(* CODESYS project Hand_Grab_Control_blocks.export

Project tree, tasks and I/O mapping:
  Hand_Grab_Control_blocks/
    data type Gesture_Type
    data type Grab_Command
    data type Grab_State
    data type PhysicalHandType
    function block Grab_Control [ST]
    function block Grab_Demo [ST]
    function block Hand_Gesture [ST]
    function block Hand_Gesture_Demo [ST]
*)

// Hand_Grab_Control_blocks/Gesture_Type
{attribute 'qualified_only'}
{attribute 'strict'}
TYPE Gesture_Type :
(
	Gesture_Type_None			:= 0,
	Gesture_Type_Num_1		:= 1,
	Gesture_Type_Num_2		:= 2,
	Gesture_Type_Num_3		:= 3,
	Gesture_Type_Num_4		:= 4,
	Gesture_Type_Num_5		:= 5,
	Gesture_Type_Num_6		:= 6,
	Gesture_Type_Fist			:= 10,
	Gesture_Type_Palm			:= 11,
	Gesture_Type_ThumbUp		:= 12,
	Gesture_Type_NoNoNo			:= 13,
	Gesture_Type_ComeOnBaby	:= 14,
	Gesture_Type_FingerWave		:= 15,
	Gesture_Type_Wave			:= 16,
	Gesture_Type_Nya			:= 17,
	Gesture_Type_MovObj			:= 18
);
END_TYPE

// Hand_Grab_Control_blocks/Grab_Command
TYPE Grab_Command :
STRUCT
	Tip_Angle : REAL;
	Root_Angle : REAL;
	Clamp_Angle : REAL;
END_STRUCT
END_TYPE

// Hand_Grab_Control_blocks/Grab_State
TYPE Grab_State :
STRUCT
	Tip_State : BOOL;
	Root_State : BOOL;
	Clamp_Angle : REAL;
END_STRUCT
END_TYPE

// Hand_Grab_Control_blocks/PhysicalHandType
TYPE PhysicalHandType :
(
	motor18		:= 0	// total 18 motors. 4 axis for thumb, 3 axis control 2 joints, anohter one control thumb tip joint. Other fingers has 3 axis each, each axis control 1 jonit. 2 axis for each wrist joint.
	, motor17	:= 10	// total 17 motors, each axis control 1 joint.
);
END_TYPE

// Hand_Grab_Control_blocks/Grab_Control
FUNCTION_BLOCK Grab_Control
VAR_INPUT
	Enable : BOOL;
	OverFeed : INT;
	Grab : Grab_Command;
	GrabFirstAxis : BYTE;
	GrabLastAxis : BYTE;
	GrabAxisAllowToMov : ARRAY [0..2] OF BOOL;
END_VAR
VAR_OUTPUT
	Done : BOOL;
	isMoving : BOOL;
	Error : BOOL;
	Err_Message : Error_Message;
	MinClampAng : REAL;
	MaxClampAng : REAL;
	MinRootAng : REAL;
	MaxRootAng : REAL;
	MinTipAng : REAL;
	MaxTipAng : REAL;
END_VAR
VAR
	state : INT := 0;
	i : INT;
	//movment settings
	Finger_Movement: MultiAxisABSMove;
	MultiMov_for_counter : INT;
	Give_Finger_Pos_Counter : INT;
	GivHandPos : ARRAY [0..255] OF REAL;
	handVel : REAL := 402;	// 402 = 67rpm
	handAcc : REAL := 4020;
	handJerk : REAL := 40200;
	givenVel, givenAcc, givenJerk : REAL;
	ArrayTotalNum : INT;
	ArrayFirstRow : INT;
	AxisAllowToMov : ARRAY [0..255] OF BOOL;
	faxis: BYTE;	// first finge axis number
	laxis : BYTE;	// last finger axis number
	
	// grab pos
	g_grab: ARRAY [0..32] OF REAL;
	
	// max degree for every motor
	grab_angle_min : REAL := 0;
	grab_angle_max : REAL := -75; //BASE
	
	Root_min : REAL := 0;
	Root_max : REAL := -138; //TURN
	
	Tip_min : REAL := 0;
	Tip_max : REAL := -86; //ROTAR
	
	// debug
	mid_0_max: REAL;
	mid_0_min: REAL;
	
	clamp : Value_Clamp;
	_ov: REAL;
END_VAR

MinClampAng := grab_angle_min;
MaxClampAng := grab_angle_max;
MinRootAng := Root_min;
MaxRootAng := Root_max;
MinTipAng := Tip_min;
MaxTipAng := Tip_max;

IF NOT Enable AND state > 0 THEN
	state := 0;
END_IF

_ov := overfeed;
IF _ov > 100 THEN
	_ov := 100;
ELSIF _ov < 1 THEN
	_ov := 1;
END_IF

Finger_Movement(firstAuxAxisNum := faxis, LastAuxAxisNum := laxis, enable := state > 0);
CASE state OF
	-30:
		error := TRUE;
		Err_Message := error_message.Err_AuxAxis_Movement_Block_err;
	-10:
	(*
		IF ReadCurrentPos.ErrorID THEN
			
		END_IF
	*)
		error := TRUE;
		Err_Message := error_message.Err_AuxAxis_Movement_Cannot_read_virture_robot_position;
	-1:
		error := TRUE;
		// can not handle more than three axis
		
	0:
		Done := error := FALSE;
		Err_Message := error_message.Err_None;
		
		IF Enable THEN
			faxis := GrabFirstAxis;
			laxis := GrabLastAxis;
			IF (laxis - faxis) <= 2 THEN
				state := 10;
			ELSE
				state := -1;
			END_IF
		END_IF

	10:	//initialize
	
		// set position
		
		// clamp Angle
		clamp(current := Grab.Clamp_Angle, first_value := grab_angle_min, second_value := grab_angle_max, newV => g_grab[0]);
		
		// clamp Root_Angle
		clamp(current := Grab.Root_Angle, first_value := Root_min, second_value := Root_max, newV => g_grab[1]);
		
		// clamp Tip_Angle
		clamp(current := Grab.Tip_Angle, first_value := Tip_min, second_value := Tip_max, newV => g_grab[2]);
		
		
		// asign value for hand movment block
		Give_Finger_Pos_Counter := 0;
		FOR MultiMov_for_counter := faxis TO laxis DO
			AxisAllowToMov[MultiMov_for_counter] := GrabAxisAllowToMov[MultiMov_for_counter - faxis];
			GivHandPos[MultiMov_for_counter] := g_grab[Give_Finger_Pos_Counter];
			Give_Finger_Pos_Counter := Give_Finger_Pos_Counter + 1;
		END_FOR
		Finger_Movement(Execute:=FALSE);
		
		givenVel := handVel * (_ov/100.0);
		givenAcc := handAcc * (_ov/100.0);
		givenJerk := handJerk * (_ov/100.0);

		State := 20;
	20:
		Finger_Movement(execute := TRUE, Axis_Mov_Indicator := AxisAllowToMov, axis_mov_pos := GivHandPos
			, vel := givenVel, acc :=givenAcc, dec := givenAcc, jerk := givenJerk, MoveMethod := 10);
		//Finger_Movement(AxesGroup:=0, Execute:=TRUE, Position:=Pos_For_Hand_Block, Settings:=Set1, active => isMoving);
		
		IF Finger_Movement.Done THEN
			Finger_Movement(Execute:=FALSE);
			done := TRUE;
			state := 50;
		ELSIF Finger_Movement.Error THEN
			state := -30;
		END_IF
	50:
			done := TRUE;
END_CASE
// end of the program

END_FUNCTION_BLOCK

// Hand_Grab_Control_blocks/Grab_Demo
FUNCTION_BLOCK Grab_Demo
VAR_INPUT
	enable :BOOL;
	internal_hand_enable : BOOL;
	startMov :BOOL;
	ovr : INT;
	GrabFirstAxis : BYTE;
	GrabLastAxis : BYTE;
	GrabAxisAllowToMov : ARRAY [0..2] OF BOOL;
END_VAR

VAR_OUTPUT
	IsEnabled : BOOL;
	IsMoving : BOOL;
	err : BOOL;
	err_message : error_message;
END_VAR

VAR
	
	// state control
	cycleState : INT;	// state machine
	cycleCounter : INT;	// counte how many time already been done
	start_cycle : INT := -1;	// start cycle from a number
	total_cycle_time : INT := 23; //	max cycle time
	cycleTimer : ton;
	cycleDelayTime : TIME := T#0MS;	// delay time between every gesture
	
	// hand powerOn
	powerHand : BOOL;
	powerOnHand : AuxAxis_PowerOn;
	_enabled : BOOL;
	
	// gestrure mov block
	GrabMov : Grab_Control;
	GrabCmd : grab_command;
	_GrabCmdEmpt : grab_command;
END_VAR


//err
IF powerOnHand.Error OR GrabMov.Error THEN
	err := TRUE;
	IF powerOnHand.Error THEN
		err_message := powerOnHand.Err_Message;
	ELSIF GrabMov.Error THEN
		err_message := GrabMov.Err_Message;
	END_IF
ELSE
	err := FALSE;
	err_message := error_message.Err_None;
END_IF

// enable hand
IF internal_hand_enable THEN
	powerOnHand(enable := enable);
	_enabled := IsEnabled := powerOnHand.Done;
END_IF

IF _enabled AND NOT internal_hand_enable THEN
	powerOnHand(enable := internal_hand_enable);
	_enabled := IsEnabled := powerOnHand.Done;
END_IF

IF NOT enable THEN
	cycleState := 0;
	isMoving := FALSE;
	cycleTimer(in := FALSE);	// reset timer
	GrabMov(Enable := FALSE);	// reset movement block
END_IF

CASE cycleState OF
	0: 
		// if block is enabled and order to move and (manager by internal power or by external power)
		IF enable AND startMov AND (NOT internal_hand_enable OR _enabled) THEN
			GrabCmd.Root_Angle := GrabMov.minRootAng;	// all open
			GrabCmd.Tip_Angle := GrabMov.minTipAng;
			GrabCmd.Clamp_Angle := GrabMov.minClampAng;
			
			cycleCounter := start_cycle;	// set counter to start_cycle
			cycleState := 10;
		END_IF
	10:
		GrabMov(Enable := TRUE, overfeed := ovr,Grab := GrabCmd, isMoving => isMoving
				, GrabFirstAxis := GrabFirstAxis, GrabLastAxis:= GrabLastAxis, GrabAxisAllowToMov:= GrabAxisAllowToMov);
		
		IF NOT startMov THEN
			GrabMov(Enable := FALSE);
			cycleState := 0;
		END_IF
		IF GrabMov.Done THEN
			cycleTimer(in := TRUE, pt:= cycleDelayTime);	// start timer for delay
			IF cycleTimer.Q THEN	// time reach
				cycleCounter := cycleCounter + 1;	// done and self add for next gesture
				cycleTimer(in := FALSE);	// reset timer
				GrabMov(Enable := FALSE);	// reset movement block
				
				IF cycleCounter <= total_cycle_time THEN
					IF cycleCounter <= 5 THEN	// first movement, root as clamp
						IF (cycleCounter MOD 2) = 1 THEN
							GrabCmd.Root_Angle := GrabMov.minRootAng;
						ELSE
							GrabCmd.Root_Angle := GrabMov.MaxRootAng;
						END_IF
					ELSIF cycleCounter <= 11 THEN	// second movement, show tip movement
						IF (cycleCounter MOD 2) = 1 THEN
							GrabCmd.Tip_Angle := GrabMov.MinTipAng;
						ELSE
							GrabCmd.Tip_Angle := GrabMov.MaxTipAng;
						END_IF
					ELSIF cyclecounter <= 17 THEN	// second movement, tip as clamp
							GrabCmd.Root_Angle := GrabMov.MaxRootAng/2;
						IF (cycleCounter MOD 2) = 1 THEN
							GrabCmd.Tip_Angle := GrabMov.MinTipAng;
						ELSE
							GrabCmd.Tip_Angle := GrabMov.MaxTipAng;
						END_IF
					ELSIF cyclecounter <= 23 THEN	// third movement, show clamp angle
						GrabCmd.Root_Angle := GrabMov.minRootAng;
						GrabCmd.Tip_Angle := GrabMov.minTipAng;
						IF (cycleCounter MOD 2) = 1 THEN;
							GrabCmd.Clamp_Angle := GrabMov.MinClampAng;
						ELSE
							GrabCmd.Clamp_Angle := GrabMov.MaxClampAng;
						END_IF
					ELSIF cyclecounter <= 24 THEN	// fouth movement, tip as clamp in another clamp angle
					END_IF
					cycleState := 10;	// if not reach total number then go back keep do next gesture
				ELSE
					cycleState := 0;	// if reach maximum then go back beginning
				END_IF
			END_IF
		END_IF
END_CASE

END_FUNCTION_BLOCK

// Hand_Grab_Control_blocks/Hand_Gesture
FUNCTION_BLOCK Hand_Gesture
VAR_INPUT
	Enable : BOOL;
	OverFeed : INT;
	Gesture : Gesture_Type;
	HandType : PhysicalHandType;	
	HandFirstAxis : BYTE;
	HandLastAxis : BYTE;
	HandAxisAllowToMov : ARRAY [0..17] OF BOOL;
END_VAR
VAR_OUTPUT
	Done : BOOL;
	isMoving : BOOL;
	Error : BOOL;
	Err_Message : Error_Message;
END_VAR
VAR
	_enb : BOOL;
	state : INT := 0;
	i : INT;
	//movment settings
	_ov : REAL;
	FingerMovPos: ARRAY [1..32] OF REAL;
	SecFingerMovPos: ARRAY [1..32] OF REAL;
	ThdFingerMovPos: ARRAY [1..32] OF REAL;
	CycleMovTimes : INT := 1;
	CycleMovDone : BOOL;
	
	CycleFingerMovPos: ARRAY [0..20] OF ARRAY[1..32] OF REAL;	
	DelayTimer : ton;
	DelayTime : ARRAY [0..20] OF TIME;
	readyToMov : BOOL;
	G_MovObj_Muilt : INT;
	
	MultisingleMov : MultiAxisABSMove;
	MultiMov_for_counter : INT;
	Give_Finger_Pos_Counter : INT;
	GivHandPos : ARRAY [0..255] OF REAL;
	handVel : REAL := 402;	// 402 = 67rpm
	handAcc : REAL := 4020;
	handJerk : REAL := 40200;
	givenVel, givenAcc, givenJerk : REAL;
	ArrayTotalNum : INT;
	ArrayFirstRow : INT;
	ReadTorque : ARRAY [0..255] OF ArcaLibrary.MCAT_ReadAxisMeasures;
	ReadTorque_For : INT;
	HandAxisTorqueValue_Sum : ARRAY [0..255] OF REAL;
	HandAxisTorqueValue_Raw : ARRAY [0..255] OF REAL;
	HandAxisTorqueValue_Smooth: ARRAY [0..255] OF REAL;
	TorqueSmoothTime : TIME := T#2S;
	TorqueSmoothTimer : ton;
	TorqueSmoothLoopTime : BYTE;
	// gesture pos
	g_RestPos: ARRAY [1..32] OF REAL;
	g_one: ARRAY [1..32] OF REAL;
	g_two: ARRAY [1..32] OF REAL;
	g_three: ARRAY [1..32] OF REAL;
	g_four: ARRAY [1..32] OF REAL;
	g_five: ARRAY [1..32] OF REAL;
	g_six: ARRAY [1..32] OF REAL;
	g_plam: ARRAY [1..32] OF REAL;
	g_fist: ARRAY [1..32] OF REAL;
	g_thumbUp: ARRAY [1..32] OF REAL;
	
	// max degree for every motor
	wrist_0_min : REAL := 0;
	wrist_0_max : REAL := 58;
	wrist_1_min : REAL := 0;
	wrist_1_max : REAL := 58;
	
	// axis 0 to axis 2
	thumb_group_pos_0 : ARRAY[0..2] OF REAL := [000, 005, 002];		// thump relex and thump tip open
	thumb_group_pos_1 : ARRAY[0..2] OF REAL := [000, 078, 002];		// thump relex and thump tip close	// this has been used in gesture fingerwave
	thumb_group_pos_2 : ARRAY[0..2] OF REAL := [120, 005, 073];		// thumb close and thump tip open	// this has been assigned to most case when thumb need to close
	thumb_group_pos_3 : ARRAY[0..2] OF REAL := [120, 078, 073];		// thumb close and thump tip close
	thumb_3_min : REAL := 0;
	thumb_3_max : REAL := 5;
	(*
	thumb_0_min : REAL := 0;
	thumb_0_max : REAL := 120;
	thumb_1_min : REAL := 5;
	thumb_1_max : REAL := 78;
	thumb_2_min : REAL := 2;
	thumb_2_max : REAL := 73;
	*)
	
	index_0_min : REAL := 0;
	index_0_max : REAL := 20;
	index_1_min : REAL := 2;
	index_1_max : REAL := 74;
	index_2_min : REAL := 1;
	index_2_max : REAL := 87;
		
	mid_0_min : REAL := 0;
	mid_0_max : REAL := 15;
	mid_1_min : REAL := 3;
	mid_1_max : REAL := 66;
	mid_2_min : REAL := 2;
	mid_2_max : REAL := 68;
			
	ring_0_min : REAL := 0;
	ring_0_max : REAL := 10;
	ring_1_min : REAL := 2;
	ring_1_max : REAL := 53;
	ring_2_min : REAL := 2;
	ring_2_max : REAL := 68;
		
	little_0_min : REAL :=0;
	little_0_max : REAL := 20;
	little_1_min : REAL := 3;
	little_1_max : REAL := 81;
	little_2_min : REAL := 1;
	little_2_max : REAL := 78;
	
	// debug
	//temp_HandType : PhysicalHandType := motor18;
	AxisAllowToMov : ARRAY [0..255] OF BOOL;
	faxis: BYTE;	// first finge axis number
	laxis : BYTE;	// last finger axis number
END_VAR

IF NOT Enable THEN
	IF _enb THEN
		_enb := done := error := FALSE;
		Err_Message := error_message.Err_None;
		state := 0;
		MultisingleMov (enable := FALSE);
		FOR readtorque_for := faxis TO laxis DO
			ReadTorque[readtorque_for](Axis := readtorque_for, Enable := FALSE);
		END_FOR
	END_IF
	RETURN;
END_IF
IF NOT _enb THEN
	_enb := TRUE;
	faxis := HandFirstAxis;	// give initialize value from globe value
	laxis := HandLastAxis;
	FOR MultiMov_for_counter := faxis TO laxis DO
		AxisAllowToMov[MultiMov_for_counter] := HandAxisAllowToMov[MultiMov_for_counter - faxis];
	END_FOR
	TorqueSmoothTimer(in := FALSE);
END_IF

_ov := overfeed;
IF _ov > 100 THEN
	_ov := 100;
ELSIF _ov < 1 THEN
	_ov := 1;
END_IF

givenVel := handVel * (_ov/100.0);
givenAcc := handAcc * (_ov/100.0);
givenJerk := handJerk * (_ov/100.0);

// read hand axis torque and smooth in time
TorqueSmoothTimer(in := TRUE, pt := TorqueSmoothTime);
IF TorqueSmoothTimer.Q THEN
	FOR readtorque_for := faxis TO laxis DO
		IF AxisAllowToMov[readtorque_for] THEN
			HandAxisTorqueValue_Smooth[readtorque_for] 
				:= HandAxisTorqueValue_Sum [readtorque_for] / TorqueSmoothLoopTime;
			HandAxisTorqueValue_Sum[readtorque_for] := 0;
		END_IF
	END_FOR
	TorqueSmoothLoopTime := 0;
	TorqueSmoothTimer(in := FALSE);
END_IF

FOR readtorque_for := faxis TO laxis DO	// read current torque
	IF AxisAllowToMov[readtorque_for] THEN
		ReadTorque[readtorque_for](Axis := readtorque_for, Enable := TRUE
			, Torque => HandAxisTorqueValue_Raw [readtorque_for]);
		HandAxisTorqueValue_Sum[readtorque_for] 
			:= HandAxisTorqueValue_Sum[readtorque_for] + HandAxisTorqueValue_Raw [readtorque_for];
	END_IF
END_FOR
TorqueSmoothLoopTime := TorqueSmoothLoopTime + 1;

MultisingleMov(firstAuxAxisNum := faxis, LastAuxAxisNum := laxis, enable := Enable);
CASE state OF
	-50:
		error := TRUE;
	-40:
		error := TRUE;
		Err_Message := error_message.Err_Gesture_Type_Cycle_mov_block_err;
	-30:
		error := TRUE;
		Err_Message := error_message.Err_AuxAxis_Movement_Block_err;
	-20:
		error := TRUE;
		Err_Message := error_message.Err_Gesture_Type_Hand_Pos_Not_Given;
	-10:
	(*
		IF ReadCurrentPos.ErrorID THEN
			
		END_IF
	*)
		error := TRUE;
		Err_Message := error_message.Err_AuxAxis_Movement_Cannot_read_virture_robot_position;
		
	0:
		IF Enable THEN
			IF Gesture <> Gesture_Type.Gesture_Type_none THEN
				state := 10;
			ELSE 
				state := -20;
			END_IF
		END_IF

	10:	//initialize
	
		// set hand pos to relax position
		g_RestPos[01] := thumb_group_pos_0[0];	//thumb_0_min;
		g_RestPos[02] := thumb_group_pos_0[1];	//thumb_1_min;
		g_RestPos[03] := thumb_group_pos_0[2];	//thumb_2_min;
		g_RestPos[04] := thumb_3_min;
		g_RestPos[05] := index_0_min;
		g_RestPos[06] := (index_1_max - index_1_min)/2 + index_1_min;
		g_RestPos[07] := (index_2_max - index_2_min)/2 + index_2_min;
		g_RestPos[08] := mid_0_min;
		g_RestPos[09] := (mid_1_max - mid_1_min)/2 + mid_1_min;
		g_RestPos[10] := (mid_2_max - mid_2_min)/2 + mid_2_min;
		g_RestPos[11] := ring_0_min;
		g_RestPos[12] := (ring_1_max - ring_1_min)/2 + ring_1_min;
		g_RestPos[13] := (ring_2_max - ring_2_min)/2 + ring_2_min;
		g_RestPos[14] := little_0_min;
		g_RestPos[15] := (little_1_max - little_1_min)/2 + little_1_min;
		g_RestPos[16] := (little_2_max - little_2_min)/2 + little_2_min;
		g_RestPos[17] := wrist_0_min;
		g_RestPos[18] := wrist_1_min;
		
		
		//one
		g_one[01]		:= thumb_group_pos_2[0];	//thumb_0_max;		//	thumb 0
		g_one[02]		:= thumb_group_pos_2[1];	//thumb_1_max;		//	thumb 1
		g_one[03]		:= thumb_group_pos_2[2];	//thumb_2_max;		//	thumb 2
		g_one[04] 		:= thumb_3_max;
		g_one[05] 		:= g_RestPos[05];	//	index 0
		g_one[06]		:= index_1_min;		//	index 1
		g_one[07]		:= index_2_min;		//	index 2
		g_one[08] 		:= g_RestPos[08];	//	mid 0
		g_one[09]		:= mid_1_max;		//	mid 1
		g_one[10]		:= mid_2_max;		//	mid 2
		g_one[11] 		:= g_RestPos[11];	//	ring 0
		g_one[12]		:= ring_1_max;		//	ring 1
		g_one[13]		:= ring_2_max;		//	ring 2
		g_one[14] 		:= g_RestPos[14];	//	little 0
		g_one[15]		:= little_1_max;	//	little 1
		g_one[16]		:= little_2_max;	//	little 2
		g_one[17]		:= g_RestPos[17];	// wrist 0
		g_one[18]		:= g_RestPos[18];	// wrist 1
		
		
		// two
		g_two[01]		:= thumb_group_pos_2[0];	//thumb_0_max;	//	thumb 0
		g_two[02]		:= thumb_group_pos_2[1];	//thumb_1_max;	//	thumb 1
		g_two[03]		:= thumb_group_pos_2[2];	//thumb_2_max;	//	thumb 2
		g_two[04] 		:= thumb_3_max;
		g_two[05]		:= g_RestPos[05];	//	index 0
		g_two[06]		:= index_1_min;		//	index 1
		g_two[07]		:= index_2_min;		//	index 2
		g_two[08]		:= g_RestPos[08];	//	mid 0
		g_two[09]		:= mid_1_min;		//	mid 1
		g_two[10]		:= mid_2_min;		//	mid 2
		g_two[11]		:= g_RestPos[11];	//	ring 0
		g_two[12]		:= ring_1_max;		//	ring 1
		g_two[13]		:= ring_2_max;		//	ring 2
		g_two[14]		:= g_RestPos[14];	//	little 0
		g_two[15]		:= little_1_max;	//	little 1
		g_two[16]		:= little_2_max;	//	little 2
		g_two[17]		:= g_RestPos[17];	// wrist 0
		g_two[18]		:= g_RestPos[18];	// wrist 1
		
		//three
		g_three[01]		:= thumb_group_pos_2[0];	//thumb_0_max;	//	thumb 0
		g_three[02]		:= thumb_group_pos_2[1];	//thumb_1_max;	//	thumb 1
		g_three[03]		:= thumb_group_pos_2[2];	//thumb_2_max;	//	thumb 2
		g_three[04] 	:= thumb_3_max;
		g_three[05]		:= g_RestPos[05];	//	index 0
		g_three[06]		:= index_1_min;		//	index 1
		g_three[07]		:= index_2_min;		//	index 2
		g_three[08]		:= g_RestPos[08];	//	mid 0
		g_three[09]		:= mid_1_min;		//	mid 1
		g_three[10]		:= mid_2_min;		//	mid 2
		g_three[11]		:= g_RestPos[11];	//	ring 0
		g_three[12]		:= ring_1_min;		//	ring 1
		g_three[13]		:= ring_2_min;		//	ring 2
		g_three[14]		:= g_RestPos[14];	//	little 0
		g_three[15]		:= little_1_max;	//	little 1
		g_three[16]		:= little_2_max;	//	little 2
		g_three[17]		:= g_RestPos[17];	// wrist 0
		g_three[18]		:= g_RestPos[18];	// wrist 1
		
		
		//four
		g_four[01]		:= thumb_group_pos_2[0];	//thumb_0_max;	//	thumb 0
		g_four[02]		:= thumb_group_pos_2[1];	//thumb_1_max;	//	thumb 1
		g_four[03]		:= thumb_group_pos_2[2];	//thumb_2_max;	//	thumb 2
		g_four[04] 		:= thumb_3_max;
		g_four[05]		:= g_RestPos[05];	//	index 0
		g_four[06]		:= index_1_min;		//	index 1
		g_four[07]		:= index_2_min;		//	index 2
		g_four[08]		:= g_RestPos[08];	//	mid 0
		g_four[09]		:= mid_1_min;		//	mid 1
		g_four[10]		:= mid_2_min;		//	mid 2
		g_four[11]		:= g_RestPos[11];	//	ring 0
		g_four[12]		:= ring_1_min;		//	ring 1
		g_four[13]		:= ring_2_min;		//	ring 2
		g_four[14]		:= g_RestPos[14];	//	little 0
		g_four[15]		:= little_1_min;	//	little 1
		g_four[16]		:= little_2_min;	//	little 2
		g_four[17]		:= g_RestPos[17];	// wrist 0
		g_four[18]		:= g_RestPos[18];	// wrist 1
		
		
		//five
		g_five[01]		:= thumb_group_pos_0[0];	//thumb_0_min;	//	thumb 0
		g_five[02]		:= thumb_group_pos_0[1];	//thumb_1_min;	//	thumb 1
		g_five[03]		:= thumb_group_pos_0[2];	//thumb_2_min;	//	thumb 2
		g_five[04] 		:= thumb_3_min;
		g_five[05]		:= g_RestPos[05];	//	index 0
		g_five[06]		:= index_1_min;		//	index 1
		g_five[07]		:= index_2_min;		//	index 2
		g_five[08]		:= g_RestPos[08];	//	mid 0
		g_five[09]		:= mid_1_min;		//	mid 1
		g_five[10]		:= mid_2_min;		//	mid 2
		g_five[11]		:= g_RestPos[11];	//	ring 0
		g_five[12]		:= ring_1_min;		//	ring 1
		g_five[13]		:= ring_2_min;		//	ring 2
		g_five[14]		:= g_RestPos[14];	//	little 0
		g_five[15]		:= little_1_min;	//	little 1
		g_five[16]		:= little_2_min;	//	little 2
		g_five[17]		:= g_RestPos[17];	// wrist 0
		g_five[18]		:= g_RestPos[18];	// wrist 1
		
		
		//six
		g_six[01]		:= thumb_group_pos_0[0];	//thumb_0_min;	//	thumb 0
		g_six[02]		:= thumb_group_pos_0[1];	//thumb_1_min;	//	thumb 1
		g_six[03]		:= thumb_group_pos_0[2];	//thumb_2_min;	//	thumb 2
		g_six[04]		:= thumb_3_min;
		g_six[05]		:= g_RestPos[05];	//	index 0
		g_six[06]		:= index_1_max;		//	index 1
		g_six[07]		:= index_2_max;		//	index 2
		g_six[08]		:= g_RestPos[08];
		g_six[09]		:= mid_1_max;	//	mid 1
		g_six[10]		:= mid_2_max;	//	mid 2
		g_six[11]		:= g_RestPos[11];
		g_six[12]		:= ring_1_max;	//	ring 1
		g_six[13]		:= ring_2_max;	//	ring 2
		g_six[14]		:= g_RestPos[14];
		g_six[15]		:= little_1_min;	//	little 1
		g_six[16]		:= little_2_min;	//	little 2
		g_six[17]		:= g_RestPos[17];	// wrist 0
		g_six[18]		:= g_RestPos[18];	// wrist 1
		
		
		//plam
		g_plam[01]		:= thumb_group_pos_0[0];	//thumb_0_min;	//	thumb 0
		g_plam[02]		:= thumb_group_pos_0[1];	//thumb_1_min;	//	thumb 1
		g_plam[03]		:= thumb_group_pos_0[2];	//thumb_2_min;	//	thumb 2
		g_plam[04]		:= thumb_3_min;
		g_plam[05]		:= g_RestPos[05];
		g_plam[06]		:= index_1_min;	//	index 1
		g_plam[07]		:= index_2_min;	//	index 2
		g_plam[08]		:= g_RestPos[08];
		g_plam[09]		:= mid_1_min;	//	mid 1
		g_plam[10]		:= mid_2_min;	//	mid 2
		g_plam[11]		:= g_RestPos[11];
		g_plam[12]		:= ring_1_min;	//	ring 1
		g_plam[13]		:= ring_2_min;	//	ring 2
		g_plam[14]		:= g_RestPos[14];
		g_plam[15]		:= little_1_min;	//	little 1
		g_plam[16]		:= little_2_min;	//	little 2
		g_plam[17]		:= g_RestPos[17];	// wrist 0
		g_plam[18]		:= g_RestPos[18];	// wrist 1
		
		
		//fist
		g_fist[01]		:= thumb_group_pos_2[0];	//thumb_0_max;	//	thumb 0
		g_fist[02]		:= thumb_group_pos_2[1];	//thumb_1_max;	//	thumb 1
		g_fist[03]		:= thumb_group_pos_2[2];	//thumb_2_max;	//	thumb 2
		g_fist[04]		:= thumb_3_max;
		g_fist[05]		:= g_RestPos[05];
		g_fist[06]		:= index_1_max;	//	index 1
		g_fist[07]		:= index_2_max;	//	index 2
		g_fist[08]		:= g_RestPos[08];
		g_fist[09]		:= mid_1_max;	//	mid 1
		g_fist[10]		:= mid_2_max;	//	mid 2
		g_fist[11]		:= g_RestPos[11];
		g_fist[12]		:= ring_1_max;	//	ring 1
		g_fist[13]		:= ring_2_max;	//	ring 2
		g_fist[14]		:= g_RestPos[14];
		g_fist[15]		:= little_1_max;	//	little 1
		g_fist[16]		:= little_2_max;	//	little 2
		g_fist[17]		:= g_RestPos[17];	// wrist 0
		g_fist[18]		:= g_RestPos[18];	// wrist 1
		
		
		//thumb up
		g_thumbUp[01]		:= thumb_group_pos_0[0];	//thumb_0_min;	//	thumb 0
		g_thumbUp[02]		:= thumb_group_pos_0[1];	//thumb_1_min;	//	thumb 1
		g_thumbUp[03]		:= thumb_group_pos_0[2];	//thumb_2_min;	//	thumb 2
		g_thumbUp[04]		:= thumb_3_min;
		g_thumbUp[05]		:= g_RestPos[05];
		g_thumbUp[06]		:= index_1_max;	//	index 1
		g_thumbUp[07]		:= index_2_max;	//	index 2
		g_thumbUp[08]		:= g_RestPos[08];
		g_thumbUp[09]		:= mid_1_max;	//	mid 1
		g_thumbUp[10]		:= mid_2_max;	//	mid 2
		g_thumbUp[11]		:= g_RestPos[11];
		g_thumbUp[12]		:= ring_1_max;	//	ring 1
		g_thumbUp[13]		:= ring_2_max;	//	ring 2
		g_thumbUp[14]		:= g_RestPos[14];
		g_thumbUp[15]		:= little_1_max;	//	little 1
		g_thumbUp[16]		:= little_2_max;	//	little 2
		g_thumbUp[17]		:= g_RestPos[17];	// wrist 0
		g_thumbUp[18]		:= g_RestPos[18];	// wrist 1
		
		CycleMovTimes := 1;	// indecate the hand will move how many cycle.
		FOR i := 0 TO 10 DO
			DelayTime[i] := T#0S;
		END_FOR
		
		DelayTime[0]:= T#0S;
		CycleFingerMovPos[0] := g_RestPos;
		
		CASE Gesture OF
			Gesture_Type.Gesture_Type_none:
				state := -20;
				
			Gesture_Type.Gesture_Type_Num_1:
				SecFingerMovPos := FingerMovPos := g_one;
				
				FingerMovPos[01]	:= g_RestPos[01];	// thumb 0
				FingerMovPos[02]	:= g_RestPos[02];	// thumb 1
				FingerMovPos[03]	:= g_RestPos[03];	// thumb 2
				FingerMovPos[04]	:= g_RestPos[04];	// thumb 3
				
				CycleMovTimes := 2;
				CycleFingerMovPos[1] := FingerMovPos;
				CycleFingerMovPos[2] := SecFingerMovPos;

			Gesture_Type.Gesture_Type_Num_2:
				SecFingerMovPos := FingerMovPos := g_two;
				
				FingerMovPos[01]	:= g_RestPos[01];	// thumb 0
				FingerMovPos[02]	:= g_RestPos[02];	// thumb 1
				FingerMovPos[03]	:= g_RestPos[03];	// thumb 2
				FingerMovPos[04]	:= g_RestPos[04];	// thumb 3
				
				CycleMovTimes := 2;
				CycleFingerMovPos[1] := FingerMovPos;
				CycleFingerMovPos[2] := SecFingerMovPos;

			Gesture_Type.Gesture_Type_Num_3:
				SecFingerMovPos := FingerMovPos := g_three;
				
				FingerMovPos[01]	:= g_RestPos[01];	// thumb 0
				FingerMovPos[02]	:= g_RestPos[02];	// thumb 1
				FingerMovPos[03]	:= g_RestPos[03];	// thumb 2
				FingerMovPos[04]	:= g_RestPos[04];	// thumb 3
				
				CycleMovTimes := 2;
				CycleFingerMovPos[1] := FingerMovPos;
				CycleFingerMovPos[2] := SecFingerMovPos;

			Gesture_Type.Gesture_Type_Num_4:
				FingerMovPos := g_four;
				
				CycleFingerMovPos[1] := FingerMovPos;

			Gesture_Type.Gesture_Type_Num_5:
				FingerMovPos := g_five;
				
				CycleFingerMovPos[1] := FingerMovPos;

			Gesture_Type.Gesture_Type_Num_6:
				FingerMovPos := g_six;
				
				CycleFingerMovPos[1] := FingerMovPos;

			Gesture_Type.Gesture_Type_Fist:
				SecFingerMovPos := FingerMovPos := g_fist;
				
				FingerMovPos[01]	:= g_RestPos[01];	// thumb 0
				FingerMovPos[02]	:= g_RestPos[02];	// thumb 1
				FingerMovPos[03]	:= g_RestPos[03];	// thumb 2
				FingerMovPos[04]	:= g_RestPos[04];	// thumb 3
				
				CycleMovTimes := 2;
				CycleFingerMovPos[1] := FingerMovPos;
				CycleFingerMovPos[2] := SecFingerMovPos;
				
			Gesture_Type.Gesture_Type_Palm:
				FingerMovPos := g_plam;
				
				CycleFingerMovPos[1] := FingerMovPos;
				
			Gesture_Type.Gesture_Type_NoNoNo:
				ThdFingerMovPos := SecFingerMovPos := FingerMovPos := g_one;
				
				FingerMovPos[01]	:= g_RestPos[01];	// thumb 0
				FingerMovPos[02]	:= g_RestPos[02];	// thumb 1
				FingerMovPos[03]	:= g_RestPos[03];	// thumb 2
				FingerMovPos[04]	:= g_RestPos[04];	// thumb 3
				
				SecFingerMovPos[05] := index_0_max;
				SecFingerMovPos[17] := wrist_0_max;	// wrist 0
				
				ThdFingerMovPos[05] := -index_0_max;
				ThdFingerMovPos[17] := -wrist_0_max;	// wrist 0
				
				CycleMovTimes := 9;
				CycleFingerMovPos[1] := FingerMovPos;
				FOR i := 2 TO CycleMovTimes DO
					IF (i MOD 2) = 1 THEN
						CycleFingerMovPos[i] := SecFingerMovPos;
					ELSE
						CycleFingerMovPos[i] := ThdFingerMovPos;
					END_IF
				END_FOR
				
			Gesture_Type.Gesture_Type_ThumbUp:
				FingerMovPos := g_thumbup;
				
				CycleFingerMovPos[1] := FingerMovPos;
				
			Gesture_Type.Gesture_Type_ComeOnBaby:
			
				ThdFingerMovPos := SecFingerMovPos := FingerMovPos := g_one;
				
				FingerMovPos[01]	:= g_RestPos[01];	// thumb 0
				FingerMovPos[02]	:= g_RestPos[02];	// thumb 1
				FingerMovPos[03]	:= g_RestPos[03];	// thumb 2
				FingerMovPos[04]	:= g_RestPos[04];	// thumb 3
				
				SecFingerMovPos[06] := g_RestPos [06];
				SecFingerMovPos[07] := index_2_max;
				
				CycleMovTimes := 9;
				CycleFingerMovPos[1] := FingerMovPos;
				FOR i := 2 TO CycleMovTimes DO
					IF (i MOD 2) = 1 THEN
						CycleFingerMovPos[i] := SecFingerMovPos;
					ELSE
						CycleFingerMovPos[i] := ThdFingerMovPos;
					END_IF
				END_FOR
				
			Gesture_Type.Gesture_Type_FingerWave:
			
				ThdFingerMovPos := SecFingerMovPos := FingerMovPos := g_plam;
				
				SecFingerMovPos[01]	:= thumb_group_pos_1[00];	// thumb 0
				SecFingerMovPos[02]	:= thumb_group_pos_1[01];	// thumb 1
				SecFingerMovPos[03]	:= thumb_group_pos_1[02];	// thumb 2
				
				SecFingerMovPos[05]	:= index_0_max;	// thumb 2
				SecFingerMovPos[08]	:= mid_0_max;	// thumb 2
				SecFingerMovPos[11]	:= ring_0_max;	// thumb 2
				SecFingerMovPos[14]	:= little_0_max;	// thumb 2
				
				ThdFingerMovPos[01]	:= g_RestPos[01];	// thumb 0
				ThdFingerMovPos[02]	:= g_RestPos[02];	// thumb 1
				ThdFingerMovPos[03]	:= g_RestPos[03];	// thumb 2
				
				ThdFingerMovPos[05]	:= -index_0_max;	// thumb 2
				ThdFingerMovPos[08]	:= -mid_0_max;	// thumb 2
				ThdFingerMovPos[11]	:= -ring_0_max;	// thumb 2
				ThdFingerMovPos[14]	:= -little_0_max;	// thumb 2
				
				CycleMovTimes := 8;
				CycleFingerMovPos[1] := FingerMovPos;
				FOR i := 2 TO CycleMovTimes DO
					IF (i MOD 2) = 1 THEN
						CycleFingerMovPos[i] := SecFingerMovPos;
					ELSE
						CycleFingerMovPos[i] := ThdFingerMovPos;
					END_IF
				END_FOR
				
			Gesture_Type.Gesture_Type_Wave:
			
				SecFingerMovPos := FingerMovPos	:= g_two;
				
				FingerMovPos[17] := wrist_0_max;
				
				SecFingerMovPos[17] := -wrist_0_max;
				
				CycleMovTimes := 8;
				FOR i := 1 TO CycleMovTimes DO
					IF (i MOD 2) = 1 THEN
						CycleFingerMovPos[i] := FingerMovPos;
					ELSE
						CycleFingerMovPos[i] := SecFingerMovPos;
					END_IF
				END_FOR
					
			Gesture_Type.Gesture_Type_Nya:
			
				SecFingerMovPos := FingerMovPos	:= g_fist;
				
				FingerMovPos[18] := wrist_1_max;
				
				SecFingerMovPos[18] := - wrist_1_max;
				
				CycleMovTimes := 8;
				FOR i := 1 TO CycleMovTimes DO
					IF (i MOD 2) = 1 THEN
						CycleFingerMovPos[i] := FingerMovPos;
					ELSE
						CycleFingerMovPos[i] := SecFingerMovPos;
					END_IF
				END_FOR
				
			Gesture_Type.Gesture_Type_MovObj:
			(*
				G_MovObj_Muilt := 2;
				FingerMovPos	:= g_plam;
				SecFingerMovPos	:= g_fist;
				CycleMovTimes := 0;	// initialize
				
				CycleMovTimes := CycleMovTimes + 1;
				FingerMovPos[12] := -wrist_0_max;
				FingerMovPos[13] := wrist_1_max;
				// first mov, hand release go up left
				CycleFingerMovPos[CycleMovTimes] := FingerMovPos;
				//---
				
				CycleMovTimes := CycleMovTimes + 1;
				FingerMovPos[12] := wrist_0_max / G_MovObj_Muilt;
				FingerMovPos[13] := wrist_1_max;
				// sec mov, hand release go down left
				CycleFingerMovPos[CycleMovTimes] := FingerMovPos;
				//---
				
				CycleMovTimes := CycleMovTimes + 1;
				SecFingerMovPos[12] := wrist_0_max  / G_MovObj_Muilt;;
				SecFingerMovPos[13] := wrist_1_max;
				// third mov, hand grab at down left
				CycleFingerMovPos[CycleMovTimes] := SecFingerMovPos;
				//---
				
				CycleMovTimes := CycleMovTimes + 1;
				SecFingerMovPos[12] := -wrist_0_max;
				SecFingerMovPos[13] := wrist_1_max;
				// 4 mov, hand grab go up left
				CycleFingerMovPos[CycleMovTimes] := SecFingerMovPos;
				//---
				
				CycleMovTimes := CycleMovTimes + 1;
				SecFingerMovPos[12] := -wrist_0_max;
				SecFingerMovPos[13] := -wrist_1_max;
				// 5 mov, hand grab go up right
				CycleFingerMovPos[CycleMovTimes] := SecFingerMovPos;
				//---
				
				CycleMovTimes := CycleMovTimes + 1;
				SecFingerMovPos[12] := wrist_0_max / G_MovObj_Muilt;;
				SecFingerMovPos[13] := -wrist_1_max;
				// 6 mov, hand grab go down right
				CycleFingerMovPos[CycleMovTimes] := SecFingerMovPos;
				//---
				
				CycleMovTimes := CycleMovTimes + 1;
				FingerMovPos[12] := wrist_0_max / G_MovObj_Muilt;;
				FingerMovPos[13] := -wrist_1_max;
				// 7 mov, hand release at down right
				CycleFingerMovPos[CycleMovTimes] := FingerMovPos;
				//---
				
				CycleMovTimes := CycleMovTimes + 1;
				FingerMovPos[12] := -wrist_0_max;
				FingerMovPos[13] := -wrist_1_max;
				// 8 mov, hand release go up right
				DelayTime[CycleMovTimes] := T#3S;
				CycleFingerMovPos[CycleMovTimes] := FingerMovPos;
				//---
				
				CycleMovTimes := CycleMovTimes + 1;
				FingerMovPos[12] := wrist_0_max / G_MovObj_Muilt;;
				FingerMovPos[13] := -wrist_1_max;
				// 9 mov, hand release go down right
				CycleFingerMovPos[CycleMovTimes] := FingerMovPos;
				//---
				
				CycleMovTimes := CycleMovTimes + 1;
				SecFingerMovPos[12] := wrist_0_max / G_MovObj_Muilt;;
				SecFingerMovPos[13] := -wrist_1_max;
				// 10 mov, hand grab at down right
				CycleFingerMovPos[CycleMovTimes] := SecFingerMovPos;
				//---
				
				CycleMovTimes := CycleMovTimes + 1;
				SecFingerMovPos[12] := -wrist_0_max;
				SecFingerMovPos[13] := -wrist_1_max;
				// 11 mov, hand grab go up right
				CycleFingerMovPos[CycleMovTimes] := SecFingerMovPos;
				//---
				
				CycleMovTimes := CycleMovTimes + 1;
				SecFingerMovPos[12] := -wrist_0_max;
				SecFingerMovPos[13] := wrist_1_max;
				// 12 mov, hand grab go up left
				CycleFingerMovPos[CycleMovTimes] := SecFingerMovPos;
				//---
				
				CycleMovTimes := CycleMovTimes + 1;
				SecFingerMovPos[12] := wrist_0_max / G_MovObj_Muilt;;
				SecFingerMovPos[13] := wrist_1_max;
				// 13 mov, hand grab at down left
				CycleFingerMovPos[CycleMovTimes] := SecFingerMovPos;
				//---
				
				CycleMovTimes := CycleMovTimes + 1;
				FingerMovPos[12] := wrist_0_max / G_MovObj_Muilt;;
				FingerMovPos[13] := wrist_1_max;
				// 14 mov, hand release at down left
				CycleFingerMovPos[CycleMovTimes] := FingerMovPos;
				//---
				*)
		END_CASE
		
		
		i := 0;
		
		Give_Finger_Pos_Counter := 1;
		ArrayTotalNum := UINT_TO_INT(SIZEOF(CycleFingerMovPos)/SIZEOF(CycleFingerMovPos[1][1]));
		ArrayFirstRow := UINT_TO_INT((SIZEOF(CycleFingerMovPos)/SIZEOF(CycleFingerMovPos[1])));
		FOR MultiMov_for_counter := faxis TO laxis DO
			IF Give_Finger_Pos_Counter <= (ArrayTotalNum/ArrayFirstRow) THEN
				GivHandPos[MultiMov_for_counter] := CycleFingerMovPos[i][Give_Finger_Pos_Counter];
				Give_Finger_Pos_Counter := Give_Finger_Pos_Counter + 1;
			END_IF
		END_FOR
		MultiSingleMov(execute := FALSE);
		
		state := 40;
		
	40:
		IF (NOT enable) THEN
			State := 0;
		END_IF
		MultisingleMov(execute := TRUE, Axis_Mov_Indicator := AxisAllowToMov, axis_mov_pos := GivHandPos
			, vel := givenVel, acc :=givenAcc, dec := givenAcc, jerk := givenJerk, MoveMethod := 10);
		
		IF MultisingleMov.Done THEN
			IF DelayTime[i] > T#0S AND NOT DelayTimer.Q THEN
				DelayTimer(in := TRUE, pt := DelayTime[i]);
			ELSE
				DelayTimer(in := FALSE);
				i := i + 1;
				
				MultisingleMov(execute:= FALSE);
				Give_Finger_Pos_Counter := 1;
				FOR MultiMov_for_counter := faxis TO laxis DO
					IF Give_Finger_Pos_Counter <= (ArrayTotalNum/ArrayFirstRow) THEN
						GivHandPos[MultiMov_for_counter] := CycleFingerMovPos[i][Give_Finger_Pos_Counter];
						Give_Finger_Pos_Counter := Give_Finger_Pos_Counter + 1;
					END_IF
				END_FOR
			END_IF
		ELSIF MultisingleMov.error THEN
			state := -40;
		END_IF
		
		IF i > CycleMovTimes THEN
			state := 50;
		END_IF
	50:
		done := TRUE;
END_CASE

// end of the program

END_FUNCTION_BLOCK

// Hand_Grab_Control_blocks/Hand_Gesture_Demo
FUNCTION_BLOCK Hand_Gesture_Demo
VAR_INPUT
	enable :BOOL;
	internal_hand_enable : BOOL;
	startMov :BOOL;
	ovr : INT;
	HandFirstAxis : BYTE;
	HandLastAxis : BYTE;
	HandAxisAllowToMov : ARRAY [0..17] OF BOOL;
END_VAR
VAR_OUTPUT
	IsEnabled : BOOL;
	IsMoving : BOOL;
	Current_Gesture : Gesture_type;
	err : BOOL;
	err_message : error_message;
END_VAR

VAR
	// state control
	cycleState : INT;	// state machine
	cycleCounter : INT;	// counte how many time already been done
	start_cycle : INT := 1;	// start cycle from a number
	total_cycle_time : INT := 14; //	max cycle time
	cycleTimer : ton;
	cycleDelayTime : TIME := T#2S;	// delay time between every gesture
	
	// hand powerOn
	powerHand : BOOL;
	powerOnHand : AuxAxis_PowerOn;
	_enabled : BOOL;
	
	// gestrure mov block
	GestureMov : Hand_Gesture;
	GestureType : ARRAY [1..16] OF Gesture_type;
END_VAR

// set gesture type
GestureType[1] := Gesture_type.Gesture_Type_Num_1;
GestureType[2] := Gesture_type.Gesture_Type_Num_2;
GestureType[3] := Gesture_type.Gesture_Type_Num_3;
GestureType[4] := Gesture_type.Gesture_Type_Num_4;
GestureType[5] := Gesture_type.Gesture_Type_Num_5;
GestureType[6] := Gesture_type.Gesture_Type_Num_6;
GestureType[7] := Gesture_type.Gesture_Type_Fist;
GestureType[8] := Gesture_type.Gesture_Type_Palm;
GestureType[9] := Gesture_type.Gesture_Type_ThumbUp;
GestureType[10] := Gesture_type.Gesture_Type_ComeOnBaby;
GestureType[11] := Gesture_type.Gesture_Type_wave;
GestureType[12] := Gesture_type.Gesture_Type_nya;
GestureType[13] := Gesture_type.Gesture_Type_NoNoNo;
GestureType[14] := Gesture_type.Gesture_Type_FingerWave;

//err
IF powerOnHand.Error OR GestureMov.Error THEN
	err := TRUE;
	IF powerOnHand.Error THEN
		err_message := powerOnHand.Err_Message;
	ELSIF GestureMov.Error THEN
		err_message := GestureMov.Err_Message;
	END_IF
ELSE
	err := FALSE;
	err_message := error_message.Err_None;
END_IF

// enable hand
IF internal_hand_enable THEN
	powerOnHand(enable := enable);
	_enabled := IsEnabled := powerOnHand.Done;
END_IF

IF NOT enable THEN
	cycleState := 0;
	isMoving := FALSE;
	cycleTimer(in := FALSE);	// reset timer
	GestureMov(Enable := FALSE);	// reset movement block
END_IF

CASE cycleState OF
	0: 
		// if block is enabled and order to move and (manager by internal power or by external power)
		IF enable AND startMov AND (NOT internal_hand_enable OR _enabled) THEN
			cycleCounter := start_cycle;	// set counter to start_cycle for gesture
			cycleState := 10;
		END_IF
	10:		GestureMov(Enable := TRUE, overfeed := ovr, Gesture := Current_Gesture := GestureType[cycleCounter], isMoving => isMoving
			, HandFirstAxis := HandFirstAxis, HandLastAxis:= HandLastAxis, HandAxisAllowToMov:= HandAxisAllowToMov);

		IF GestureMov.Done THEN
			cycleTimer(in := TRUE, pt:= cycleDelayTime);	// start timer for delay
			IF cycleTimer.Q THEN	// time reach
				cycleCounter := cycleCounter + 1;	// done and self add for next gesture
				cycleTimer(in := FALSE);	// reset timer
				GestureMov(Enable := FALSE);	// reset movement block
				IF cycleCounter <= total_cycle_time THEN
					cycleState := 10;	// if not reach total number then go back keep do next gesture
				ELSE
					cycleState := 0;	// if reach maximum then go back beginning
				END_IF
			END_IF
		END_IF
		
END_CASE

END_FUNCTION_BLOCK
